Fanuc KAREL source: tpelib.kl

PROGRAM tpelib
%NOLOCKGROUP

%include tpe.klt

--hash struct
%include hash_tpeprog.klt
t_hash(hashname,TPEPROGRM,TPE_DICTIONARY_FILENAME)

VAR
  prgm_stats : ARRAY[10] OF hashname
  curr_prog : STRING[30]
  curr_line : STRING[128]
  new_prog : STRING[30]
  tpefile : FILE
  newfile : FILE

%from errors.klh %import CHK_STAT, karelError
%from pose.klh %import jpos_to_jpos6, jpos_to_jpos2
%include strings.klh
%include files.klh

%include tpe.private.klh
%include tpe.klh
%include tpe_hash.klh

-- Define TPE dictionary file
%class `TPE_DICTIONARY_FILENAME`('hash.klc','hashclass.klh','hash_tpeprog.klt')

BEGIN
END tpelib

-- *** PRIVATE ***

-- *** PUBLIC ***

-- handlers
-- ***********
ROUTINE tpe__constructor
  VAR
    empty : TPEPROGRM
    b : BOOLEAN
  BEGIN
    empty.open_id = 0 ; empty.status = 0 ;
    b = `TPE_DICTIONARY_FILENAME`__clear_table('tpelib', 'prgm_stats', empty)
  END tpe__constructor


ROUTINE tpe__destructor
  VAR
    empty  : TPEPROGRM
    b : BOOLEAN
  BEGIN
    empty.open_id = 0 ; empty.status = 0 ;
     b = `TPE_DICTIONARY_FILENAME`__clear_table('tpelib', 'prgm_stats', empty)
  END tpe__destructor


ROUTINE tpe__open
  VAR
    p_stat : TPEPROGRM
    open_id, status : INTEGER
    b : BOOLEAN
  BEGIN
    -- Open TPE program in read only
    OPEN_TPE(TPE_name, TPE_RDACC, TPE_NOREJ, open_id, status)
    --check status, abort if nessecary
    CHK_STAT(status)

    --add to hash
    p_stat.open_id = open_id
    -- set status to TPE_IS_OPEN
    -- or list the error code
    IF (status = 0) THEN
      p_stat.status = TPE_IS_OPEN
    ELSE
      p_stat.status = status
    ENDIF

    b = `TPE_DICTIONARY_FILENAME`__put(TPE_name, p_stat, 'tpelib', 'prgm_stats')
    IF NOT b THEN karelError(INVALID_INDEX, 'Could not write '+ TPE_name + ' to "prgm_stats" in TPE', ER_ABORT) ; ENDIF

    RETURN(open_id)

  END tpe__open

ROUTINE tpe__close
  VAR
    p_stat : TPEPROGRM
    status : INTEGER
    b : BOOLEAN
  BEGIN
    -- get openid if it exists
    b = `TPE_DICTIONARY_FILENAME`__get(TPE_name, p_stat, 'tpelib', 'prgm_stats')
    IF NOT b THEN karelError(TPE_UPDATE_FAILED, TPE_name + ' does not appear to be open.', ER_WARN) ; ENDIF
    --close if program foudn in log
    IF b THEN
      --close tpe program
      CLOSE_TPE (p_stat.open_id, status)
      --check status
      CHK_STAT(status)
      --remove from hash
      b = `TPE_DICTIONARY_FILENAME`__delete(TPE_name, 'tpelib', 'prgm_stats')
    ENDIF

  END tpe__close

ROUTINE tpe__delete
  VAR
    p_stat : TPEPROGRM
    upper_name : STRING[30]
    b : BOOLEAN
  BEGIN
    --if program is currently open, close it first to keep the hash consistent
    b = `TPE_DICTIONARY_FILENAME`__get(TPE_name, p_stat, 'tpelib', 'prgm_stats')
    IF b THEN
      tpe__close(TPE_name)
    ENDIF

    upper_name = to_upper(TPE_name)
    files__delete('MD:/' + upper_name + '.LS')
    files__delete('MD:/' + upper_name + '.TP')
  END tpe__delete

ROUTINE tpe__delete_pattern
  VAR
    upper_name : STRING[30]
  BEGIN
    --pattern may include the * wildcard, e.g. 'TMPS_CYLGEN*'
    --caller must ensure no matching programs are currently open via tpe__open;
    --DELETE_FILE will return a non-"not found" status for any open .TP,
    --which files__delete propagates as an abort.
    upper_name = to_upper(TPE_prefix)
    files__delete('MD:/' + upper_name + '*.LS')
    files__delete('MD:/' + upper_name + '*.TP')
  END tpe__delete_pattern

ROUTINE tpe__open_file
  VAR
    dstr : STRING[3]
  BEGIN
    curr_prog = 'MD:/'+to_upper(TPE_name)+'.LS'
    curr_line = ''

    files__open(curr_prog, 'RO', tpefile)
    dstr = ''

    --buffer until the start of the program
    WHILE dstr <> '/MN' DO
      files__read_line_ref(curr_prog, tpefile, curr_line)
      dstr = SUB_STR(curr_line,1,3)
    ENDWHILE

  END tpe__open_file

ROUTINE tpe__close_file
  BEGIN
    files__close(curr_prog, tpefile)

    curr_prog = ''
    curr_line = ''
  END tpe__close_file

ROUTINE tpe__sanitize_line
  VAR
    idx : INTEGER
  BEGIN
    --remove leading spaces
    curr_line = lstrip(curr_line)
    --find index of colon
    idx = 0
    idx = char_index(curr_line, ':')
    IF idx > 0 THEN
      curr_line = SUB_STR(curr_line, idx+1, STR_LEN(curr_line))
    ENDIF

    --remove trailing spaces
    curr_line = rstrip(curr_line)
    --assume last character is semi-colon
    IF SUB_STR(curr_line, STR_LEN(curr_line), 1) = ';' THEN
      curr_line = SUB_STR(curr_line, 1, STR_LEN(curr_line)-1)
    ENDIF

  END tpe__sanitize_line

ROUTINE tpe__get_tpeprogram
  VAR
    p_stat : TPEPROGRM
    b : BOOLEAN
  BEGIN
    --see if file is already open
    b = `TPE_DICTIONARY_FILENAME`__get(TPE_name, p_stat, 'tpelib', 'prgm_stats')
    IF NOT b THEN
      karelError(FILE_NOT_OPEN, TPE_name + ' is not open. use TPE__open to open file first.', ER_WARN)
    ENDIF

    RETURN(p_stat)
  END tpe__get_tpeprogram

  ROUTINE tpe__get_open_id
  VAR
    p_stat : TPEPROGRM
    b : BOOLEAN
  BEGIN
    --see if file is already open
    b = `TPE_DICTIONARY_FILENAME`__get(TPE_name, p_stat, 'tpelib', 'prgm_stats')
    IF NOT b THEN
      karelError(FILE_NOT_OPEN, TPE_name + ' is not open. use TPE__open to open file first.', ER_WARN)
    ENDIF

    RETURN(p_stat.open_id)
  END tpe__get_open_id

ROUTINE tpe__copy
  VAR
    status : INTEGER
  BEGIN
    COPY_TPE(TPE_name,new_name,TRUE,status)
	  CHK_STAT(status)
  END tpe__copy


-- Write to TPE files
-- *******************

ROUTINE tpe__create
  VAR
    status : INTEGER
  BEGIN
    --create new TPE file
    CREATE_TPE(name, PT_MNE_UNDEF, status)
    --if program exists delete it and try again
    IF status = TPE_PROGRAM_ALREADY_EXISTS THEN
      files__delete('MD:/'+to_upper(name)+'.LS')
      CREATE_TPE(name, PT_MNE_UNDEF, status)
    ENDIF
    CHK_STAT(status)
  END tpe__create


ROUTINE tpe__create_ls
  BEGIN
    new_prog = 'MD:/'+to_upper(name)+'.LS'
    files__open(new_prog, 'RW', newfile)

    --write program name to file
    curr_line = '/PROG ' + to_upper(name)
    files__write_line(curr_line, new_prog, newfile)
  END tpe__create_ls


ROUTINE tpe__close_ls
  BEGIN
    files__close(new_prog, newfile)
    --new_prog = ''
  END tpe__close_ls

ROUTINE tpe__pns_name
  BEGIN
    RETURN(prefix + i_to_s(number))
  END tpe__pns_name

ROUTINE tpe__ls_exists
  VAR
    ec : INTEGER
  BEGIN
    curr_prog = 'MD:/'+to_upper(TPE_Name)+'.TP'

    CLR_IO_STAT(tpefile)
    OPEN FILE tpefile('RO', curr_prog)
    ec = IO_STATUS(tpefile)

    WRITE(CR,ec)

    IF ec = 0 THEN
      CLOSE FILE tpefile
      RETURN(TRUE)
    ENDIF

    RETURN(FALSE)

  END tpe__ls_exists

ROUTINE tpe__copy_header_ls
  VAR
    dstr : STRING[3]
    status : INTEGER
  BEGIN
    --open created TPE file to read through program
    curr_prog = 'MD:/'+to_upper(TPE_Name)+'.LS'
    files__open(curr_prog, 'RO', tpefile)

    curr_line = ''
    dstr = ''

    --skip program name
    files__read_line_ref(curr_prog, tpefile, curr_line)

    --buffer until the start of the program
    WHILE dstr <> '/MN' DO
      files__read_line_ref(curr_prog, tpefile, curr_line)
      dstr = SUB_STR(curr_line,1,3)
      --Write the TPE file to the LS file up until the start of the program
      files__write_line(curr_line, new_prog, newfile)
    ENDWHILE
    --write /MN to start the program
    files__write_line('/MN', new_prog, newfile)

    --close the TPE file
    files__close(curr_prog, tpefile)
    curr_prog = ''
    curr_line = ''

  END tpe__copy_header_ls


ROUTINE tpe__write_end
  BEGIN
    files__write_line('/POS', new_prog, newfile)
    files__write_line('/END', new_prog, newfile)
  END tpe__write_end

ROUTINE tpe__write_pause
  BEGIN
    files__write_line(':  PAUSE ;', new_prog, newfile)
  END tpe__write_pause

ROUTINE tpe__write_uframe
  BEGIN
    files__write_line(':  UFRAME_NUM='+ i_to_s(num) +' ;', new_prog, newfile)
  END tpe__write_uframe

ROUTINE tpe__write_utool
  BEGIN
    files__write_line(':  UTOOL_NUM='+ i_to_s(num) +' ;', new_prog, newfile)
  END tpe__write_utool

ROUTINE tpe__write_line
  BEGIN
    files__write_line(str, new_prog, newfile)
  END tpe__write_line


--get AR variables from TPE file
--******************

-- Return int LS argument value
ROUTINE tpe__get_int_arg
  VAR
    data_type  : INTEGER
    int_value  : INTEGER
    real_value : REAL
    string_value : STRING[1]
    STATUS     : INTEGER
  BEGIN
    data_type = Type_INTEGER

    GET_TPE_PRM(reg_no, data_type, int_value, real_value, string_value, STATUS)
    IF STATUS = NOPARAM THEN
        WRITE('Parameter AR[', reg_no ,'] does not exist.')
    ENDIF
    IF data_type <> 1 THEN
      karelError(EXPECTED_INT, 'TPE argument ' + i_to_s(reg_no) + ' is not an integer', ER_ABORT)
    ENDIF
    CHK_STAT(STATUS)

    RETURN(int_value)

  END tpe__get_int_arg


-- Return real LS argument value
ROUTINE tpe__get_real_arg
  VAR
    data_type  : INTEGER
    int_value  : INTEGER
    real_value : REAL
    string_value : STRING[1]
    STATUS     : INTEGER
  BEGIN
    data_type = Type_REAL

    GET_TPE_PRM(reg_no, data_type, int_value, real_value, string_value, STATUS)
    IF (real_value = 0) AND (int_value <> 0) THEN
      real_value = int_value
    ENDIF
    IF data_type = 3  THEN
      karelError(EXPECTED_REAL, 'TPE argument ' + i_to_s(reg_no) + ' is not a number', ER_ABORT)
    ENDIF
    IF STATUS = NOPARAM THEN
        WRITE('Parameter AR[', reg_no ,'] does not exist.')
    ENDIF
    CHK_STAT(STATUS)

    RETURN(real_value)

  END tpe__get_real_arg


-- get LS string argument
ROUTINE tpe__get_string_arg
  VAR
    data_type  : INTEGER
    int_value  : INTEGER
    real_value : REAL
    string_value : STRING[32]
    STATUS     : INTEGER
  BEGIN
    data_type = Type_STRING

    GET_TPE_PRM(reg_no, data_type, int_value, real_value, string_value, STATUS)
    IF STATUS = NOPARAM THEN
        WRITE('Parameter AR[', reg_no ,'] does not exist.')
    ENDIF
    IF data_type <> 3 THEN
      karelError(INVALID_STRING, 'TPE argument ' + i_to_s(reg_no) + ' is not a string', ER_ABORT)
    ENDIF

    CHK_STAT(STATUS)

    RETURN(string_value)
  END tpe__get_string_arg

ROUTINE tpe__get_boolean_arg
  VAR
    data_type  : INTEGER
    int_value  : INTEGER
    real_value : REAL
    string_value : STRING[1]
    STATUS     : INTEGER
  BEGIN
    data_type = Type_INTEGER

    GET_TPE_PRM(reg_no, data_type, int_value, real_value, string_value, STATUS)
    IF STATUS = NOPARAM THEN
        WRITE('Parameter AR[', reg_no ,'] does not exist.')
    ENDIF
    IF data_type <> 1 THEN
      karelError(EXPECTED_INT, 'TPE argument ' + i_to_s(reg_no) + ' is not an integer', ER_ABORT)
    ENDIF
    CHK_STAT(STATUS)

    IF (int_value = 0) THEN
      RETURN(FALSE)
    ENDIF

    RETURN(TRUE)
  END tpe__get_boolean_arg

ROUTINE tpe__get_vector_arg
  VAR
    p : XYZWPR
    v : VECTOR
    STATUS : INTEGER
  BEGIN
    IF (reg_no <= 0) THEN
        WRITE TPERROR (CR, 'position register must be > 0')
    ENDIF

    p = GET_POS_REG(reg_no, STATUS, 1)
    CHK_STAT(STATUS)
    IF STATUS <> 0 THEN
        karelError(POS_REG_NOT_SET,'PR' + i_to_s(reg_no) + ' not set for vector arg.', ER_ABORT)
    ENDIF

    v.x = p.x ; v.y = p.y ; v.z = p.z ;

    RETURN(v)

  END tpe__get_vector_arg

ROUTINE tpe__parameter_exists
  VAR
    data_type  : INTEGER
    int_value  : INTEGER
    real_value : REAL
    string_value : STRING[32]
    STATUS     : INTEGER
  BEGIN
    GET_TPE_PRM(reg_no, data_type, int_value, real_value, string_value, STATUS)
    IF STATUS = NOPARAM THEN
      RETURN(FALSE)
    ELSE
      RETURN(TRUE)
    ENDIF
  END tpe__parameter_exists
